// TIA Portal V20 export
// export: Created 2025-12-01T14:57:22.9974681Z, ExportSetting None, DisplayName Totally Integrated Automation Portal, DisplayVersion V20 Update 3, DisplayName TIA Portal Openness, DisplayVersion V20 Update 3, DisplayName TIA Portal Version Control Interface, DisplayVersion V20 Update 3, DisplayName STEP 7 Professional, DisplayVersion V20 Update 3, DisplayName STEP 7 Safety, DisplayVersion V20 Update 2, DisplayName WinCC Basic/Comfort/Advanced, DisplayVersion V20 Update 3, DisplayName WinCC Professional, DisplayVersion V20 Update 3, DisplayName WinCC Unified, DisplayVersion V20 Update 3
DATA_BLOCK "DB914_Conf_Mesas_DeZona"   // DB914
{ S7_Optimized_Access := 'FALSE' }
// stored: AutoNumber false
   VAR RETAIN
      MesasDeZona { S7_SetPoint := 'True'} : Array[0.."CTE_MaxMesas", 0..4] of "ZonaPerteneceMesa";
   END_VAR
BEGIN
END_DATA_BLOCK
